(* PLC project Blank Project, Blank Blank 1.0 *)
(* stored: creationDateTime 2016-05-18T21:14:07, modificationDateTime 2018-06-25T14:34:19 *)

FUNCTION_BLOCK Temp_Conversion
  VAR_INPUT
    raw_temp : UINT;
  END_VAR
  VAR
    voltage : REAL;
    resistance : REAL;
    steinhart : REAL;
    THERMISTORNOMINAL : REAL := 10000.0;
    TEMPERATURENOMINAL : REAL := 25.0;
    BCOEFFICIENT : REAL := 3950.0;
    SERIESRESISTOR : REAL := 10000.0;
  END_VAR
  VAR_OUTPUT
    converted_temp : INT;
    voltage_out : INT;
    resistance_out : INT;
  END_VAR

            (* Calculate Voltage *)
voltage := UINT_TO_REAL(raw_temp);
voltage := voltage * 0.0001535107446;

(* Calculate Resistance *)
resistance := voltage / 10.0;
resistance := 1.0 / resistance;
resistance := resistance - 1.0;
resistance := resistance * 10000.0;


(* Calculate Steinhart *)
steinhart := resistance / THERMISTORNOMINAL; (* (R/Ro) *)
steinhart := LN(steinhart); (* ln(R/Ro) *)
steinhart := steinhart / BCOEFFICIENT; (* 1/B * ln(R/Ro) *)
steinhart := steinhart + 1.0 / (TEMPERATURENOMINAL + 273.15); (* (1/To) *)
steinhart := 1.0 / steinhart; (* Invert *)
steinhart := steinhart - 273.15; (* Convert to C *)

(* Calculate the error correction *)
steinhart := steinhart + 9.451149;
steinhart := steinhart / 0.894263;
steinhart := steinhart * 100.0; (* Multiply by 100 to get 2 decimals *)

voltage_out := REAL_TO_INT(voltage * 100.0);
resistance_out := REAL_TO_INT(resistance);
converted_temp := REAL_TO_INT(steinhart);

(*
voltage := UINT_TO_REAL(raw_temp);
voltage := 10000.0 / (65536.0 / voltage - 1.0);
voltage := voltage / 10000.0;
voltage := LN(voltage);
voltage := 1.0 / ((1.0/298.15) + (voltage * (1.0/3950.0)));
voltage := voltage - 273.15;
voltage := voltage * 100.0;
converted_temp := REAL_TO_INT(voltage);
*)

          
END_FUNCTION_BLOCK

PROGRAM My_Program
  VAR
    raw_temp AT %IW0 : UINT;
    Ref_Voltage AT %QW0 : UINT := 65535;
    converted_temp AT %QW1 : INT;
    voltage AT %QW7 : INT;
    resistance AT %QW8 : INT;
    setpoint AT %QW2 : INT := 4000;
    mode_register AT %QW4 : INT;
    heater_control AT %QW5 : INT;
    heater_man AT %QX99.0 : BOOL;
    heater_auto AT %QX99.1 : BOOL;
    heater AT %QX0.0 : BOOL;
  END_VAR
  VAR
    Temp_Conversion0 : Temp_Conversion;
  END_VAR

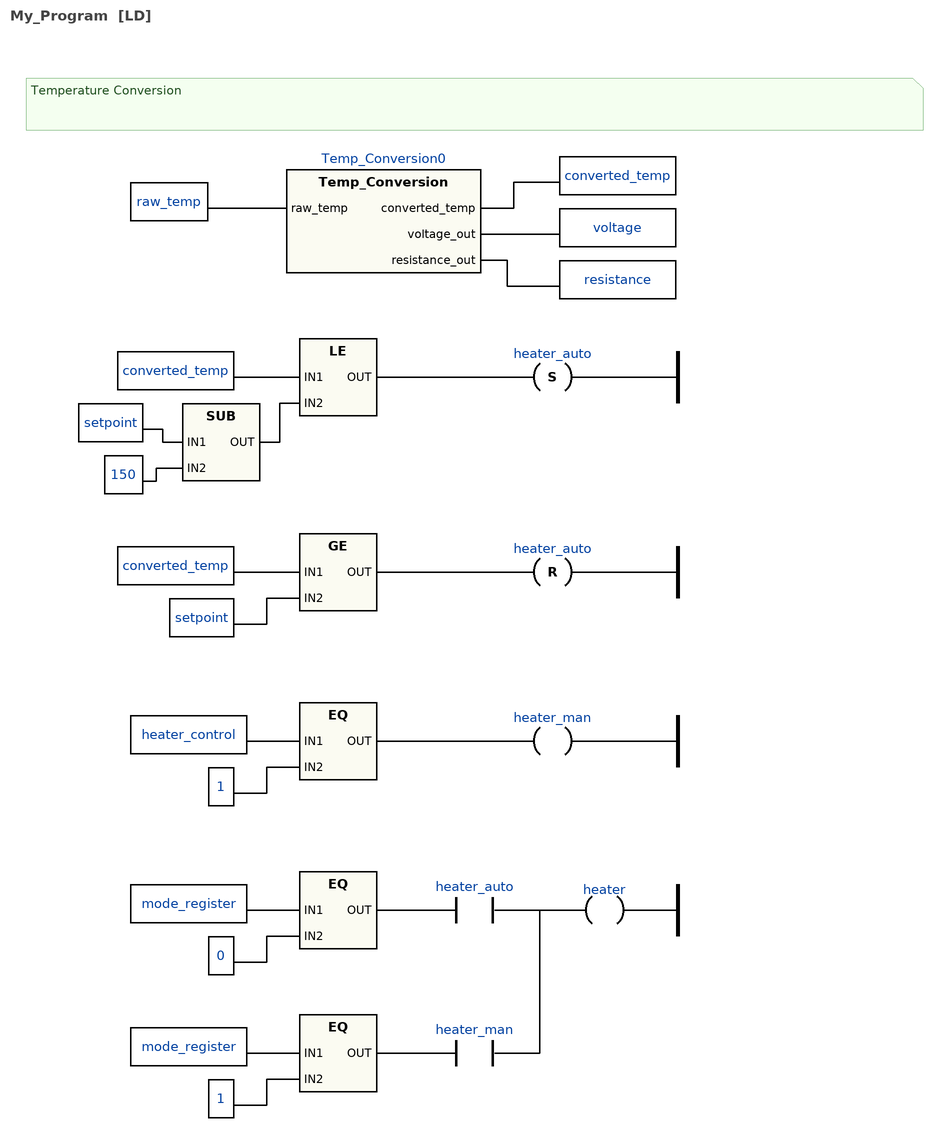
(* LD diagram, written out as Structured Text *)
(* Temperature Conversion *)
Temp_Conversion0(raw_temp := raw_temp);
converted_temp := Temp_Conversion0.converted_temp;
voltage := Temp_Conversion0.voltage_out;
resistance := Temp_Conversion0.resistance_out;
IF converted_temp <= setpoint - 150 THEN heater_auto := TRUE; END_IF;
IF converted_temp >= setpoint THEN heater_auto := FALSE; END_IF;
heater_man := heater_control = 1;
heater := mode_register = 0 AND heater_auto OR mode_register = 1 AND heater_man;
END_PROGRAM

CONFIGURATION Config0
  RESOURCE Res0 ON PLC
    TASK TaskMain(INTERVAL := T#50ms, PRIORITY := 0);
    PROGRAM Inst0 WITH TaskMain : My_Program;
  END_RESOURCE
END_CONFIGURATION
